FUNCTION_BLOCK XtsPart EXTENDS CyclicBase
VAR
	_MyInterface : Tc3_XTS_Utility.I_TcIoXtsXpuPart;
	XtsIoEnvInitialiseState : INT;
	MyModuleCount : UDINT;
	PartDriveState: Tc3_XTS_Utility.DriveState;
	_ReadyToEnable: BOOL;
	Modules : ARRAY[1..SystemParameters.MaxModulesInPart] OF I_TcIoXtsPartModule;
	ModulesCoE : ARRAY[1..SystemParameters.MaxModulesInPart] OF I_AT2xxxXtsMotor;
	f24V: ARRAY[1..SystemParameters.MaxModulesInPart] OF UINT;
	f48V: ARRAY[1..SystemParameters.MaxModulesInPart] OF UINT;
	CurrentLive : ARRAY[1..SystemParameters.MaxModulesInPart] OF DINT;
	MaxCurrent : ARRAY [1..SystemParameters.MaxModulesInPart] OF DINT;
	ModuleIndex: UDINT := 1;
	i : UINT;
END_VAR

METHOD PUBLIC  Cycle : HRESULT
VAR_INPUT
END_VAR
getModuleInfoData();

PartDriveState := _MyInterface.GetDriveState();

CASE PartDriveState OF
	DriveState.Unknown:
		_ReadyToEnable := FALSE;

	DriveState.FaultReactionActive:
		_ReadyToEnable := FALSE;

	DriveState.Fault:
		_ReadyToEnable := FALSE;

	DriveState.NotReadyToSwitchOn:
		_ReadyToEnable := FALSE;

	DriveState.SwitchOnDisabled:
		_ReadyToEnable := FALSE;

	DriveState.ReadyToSwitchOn:
		_ReadyToEnable := TRUE;

	DriveState.SwitchedOn:
		_ReadyToEnable := TRUE;

	DriveState.OperationEnabled:
		_ReadyToEnable := TRUE;

ELSE
	_ReadyToEnable := FALSE;
END_CASE
END_METHOD

METHOD PRIVATE getModuleInfoData : BOOL
VAR_INPUT
END_VAR
IF ModulesCoE[ModuleIndex].InfoData.Update() THEN
	CurrentLive[ModuleIndex]:=ModulesCoE[ModuleIndex].InfoData.OverallCurrent;
	MaxCurrent[ModuleIndex]:=ModulesCoE[ModuleIndex].InfoData.MaxOverallCurrentLast500ms;
	f24V[ModuleIndex]:= ModulesCoE[ModuleIndex].InfoData.AuxiliaryVoltage24V;
	f48V[ModuleIndex]:=ModulesCoE[ModuleIndex].InfoData.DcLinkVoltage;
	IF ModuleIndex = MyModuleCount THEN
		ModuleIndex := 1;
	ELSE
		ModuleIndex := ModuleIndex + 1;
	END_IF
END_IF
END_METHOD

METHOD Initialise : HRESULT
VAR_INPUT
END_VAR
CASE XtsIoEnvInitialiseState OF
	0:
		IF _MyInterface <> 0 THEN
			XtsIoEnvInitialiseState := 1;
		ELSE
			XtsIoEnvInitialiseState := 999;
		END_IF
	1:
		MyModuleCount := _MyInterface.GetModuleCount();
		FOR i := 1 TO UDINT_TO_UINT(MyModuleCount) DO
			Modules[i] := _MyInterface.ModuleTcIo(i);
			ModulesCoE[i] := _MyInterface.ModuleCoE(i);
		END_FOR
		XtsIoEnvInitialiseState := 2;
	2:
		XtsIoEnvInitialiseState := 3;
		FOR i := 1 TO UDINT_TO_UINT(MyModuleCount) DO
			IF NOT Modules[i].P_IsInitialized THEN
				XtsIoEnvInitialiseState := 2;
			END_IF
		END_FOR
	3:
		Initialise := 2;

END_CASE
END_METHOD

METHOD Is24VOK : HRESULT
VAR_INPUT
END_VAR
Is24VOK := 2;
FOR i := 1 TO UDINT_TO_UINT(MyModuleCount) DO
	IF f24V[i] < 20400 THEN
		Is24VOK := 1;
	END_IF
	IF f24V[i] > 28800 THEN
		Is24VOK := 1;
	END_IF
END_FOR
END_METHOD

METHOD Is48VOK : HRESULT
VAR_INPUT
END_VAR
Is48VOK := 2;
FOR i := 1 TO UDINT_TO_UINT(MyModuleCount) DO
	IF f48V[i] < 46080 THEN
		Is48VOK := 1;
	END_IF
	IF f48V[i] > 49920 THEN
		Is48VOK := 1;
	END_IF
END_FOR
END_METHOD

PROPERTY MyXtsIoEnvInterface : I_TcIoXtsXpuPart
GET
MyXtsIoEnvInterface := _MyInterface;
END_GET
SET
_MyInterface := MyXtsIoEnvInterface;
END_SET
END_PROPERTY

END_FUNCTION_BLOCK

(* stored: Version 1.1.0.1, ProductVersion 3.1.4024.12
   POU XtsPart: Id {39541d00-22ec-4750-829d-4864a624597e}, SpecialFunc None
   Method Cycle: Id {6aa26807-846b-4168-ab87-fb4c66b138eb}
   Method getModuleInfoData: Id {3efa41b4-5489-4d81-8938-0f058eef3c58}
   Method Initialise: Id {f7bcb601-a320-4f3f-bcf3-5ec4e45a7245}
   Method Is24VOK: Id {2b0cb545-a877-4023-acf7-204433c79109}
   Method Is48VOK: Id {85bd6738-1af1-443c-8d2c-d0704993fb05}
   Property MyXtsIoEnvInterface: Id {b5f6c838-c909-4a11-9656-9e449699aee4}
   Get Get: Id {249dae7e-fa2b-4c2d-a421-a33d92e9b50d}
   Set Set: Id {436f8d77-48c4-4edc-81e4-5821f3038a93} *)
